PROGRAM P_SlaveInputControl
VAR
	tempEncoder1 : LREAL := 0;
	tempEncoder11 : LREAL := 1;
END_VAR

END_PROGRAM

(* stored: Version 1.1.0.1, ProductVersion 3.1.4024.12
   POU P_SlaveInputControl: Id {484f9364-46d2-4430-a336-f7521af6b9ce}, SpecialFunc None *)
